FUNCTION_BLOCK "Sequence"   // FB18, GRAPH_PLUS
{ S7_Optimized_Access := 'TRUE' }
VERSION : 0.1
   VAR_INPUT
      OFF_SQ : Bool := false;   // Turn sequence off
      INIT_SQ : Bool := false;   // Set sequence to initial state
      ACK_EF : Bool := false;   // Acknowledge all errors and faults
      S_PREV : Bool := false;   // Output previous step in parameter S_NO
      S_NEXT : Bool := false;   // Indicate next step in parameter S_NO
      SW_AUTO : Bool := false;   // Automatic mode
      SW_TAP : Bool := false;   // Semiautomatic/switch with transition
      SW_TOP : Bool := false;   // Semiautomatic/ignore transition
      SW_MAN : Bool := false;   // Manual mode
      S_SEL : Int := 0;   // Select step to be output to S_NO
      S_ON : Bool := false;   // Activate step indicated in S_NO
      S_OFF : Bool := false;   // Deactivate step indicated S_NO
      T_PUSH : Bool := false;   // Enable transition to switch in semi automatic mode
   END_VAR
   VAR_OUTPUT
      S_NO : Int := 0;   // Step number
      S_MORE : Bool := false;   // More steps are available and can be shown in S_NO
      S_ACTIVE : Bool := false;   // Step indicated in S_NO is active
      ERR_FLT : Bool := false;   // Interlock or supervision group error
      AUTO_ON : Bool := false;   // Automatic mode is active
      TAP_ON : Bool := false;   // Semiautomatic mode/step with transition enabled
      TOP_ON : Bool := false;   // Semiautomatic mode/ignore transition enabled
      MAN_ON : Bool := false;   // Manual mode is active
   END_VAR
   VAR
      HMI_INFO : Array[0..8] of UInt;
      IF_PAR : G7_IfParPlus_V2;
      RT_DATA : G7_RTDataPlus_V2;   // Internal data area
      Trans1 : G7_TransitionPlus_V2;   // Transition structure
      Trans2 : G7_TransitionPlus_V2;   // Transition structure
      Trans3 : G7_TransitionPlus_V2;   // Transition structure
      Trans4 : G7_TransitionPlus_V2;   // Transition structure
      Trans5 : G7_TransitionPlus_V2;   // Transition structure
      idle : G7_StepPlus_V2;   // Step structure
      warmup : G7_StepPlus_V2;   // Step structure
      stabilize : G7_StepPlus_V2;   // Step structure
      Generation : G7_StepPlus_V2;   // Step structure
      cooldown : G7_StepPlus_V2;   // Step structure
      SINI : Array[0..1] of USInt;
      LSTT : Array[0..4] of USInt;
      ATAJ : Array[0..4] of USInt;
      ATAB : Array[0..4] of USInt;
      PSTT : Array[0..4] of USInt;
      NSTT : Array[0..4] of USInt;
      ASSJ : Array[0..4] of USInt;
      ASSB : Array[0..4] of USInt;
      PTTS : Array[0..4] of USInt;
      NTTS : Array[0..4] of USInt;
      SW_SQTS : Array[0..4] of USInt;
      SWITCH : Array[0..0] of USInt;
      TVX : Array[0..1] of USInt;
      TTX : Array[0..1] of USInt;
      TSX : Array[0..1] of USInt;
      S00X : Array[0..1] of USInt;
      SOFFX : Array[0..1] of USInt;
      SONX : Array[0..1] of USInt;
      SAX : Array[0..1] of USInt;
      SERRX : Array[0..5] of USInt;
      SMX : Array[0..5] of USInt;
      S0X : Array[0..5] of USInt;
      S1X : Array[0..5] of USInt;
      IL_ALARM_INST : Program_Alarm;
      SUP_ALARM_INST : Program_Alarm;
      STEP_TIME_ALARM_INST : Program_Alarm;
      IEC_TIMER_INST : IEC_TIMER;
      TRANSACTION_FLAG : Bool := false;
   END_VAR
   // SINI[0] := 2;
   // LSTT[0] := 255;
   // LSTT[1] := 255;
   // LSTT[2] := 255;
   // LSTT[3] := 255;
   // ATAJ[1] := 1;
   // ATAJ[2] := 2;
   // ATAJ[3] := 3;
   // ATAJ[4] := 4;
   // ATAB[1] := 1;
   // ATAB[2] := 2;
   // ATAB[3] := 3;
   // ATAB[4] := 4;
   // PSTT[1] := 1;
   // PSTT[2] := 2;
   // PSTT[3] := 3;
   // PSTT[4] := 4;
   // NSTT[0] := 1;
   // NSTT[1] := 2;
   // NSTT[2] := 3;
   // NSTT[3] := 4;
   // ASSJ[1] := 1;
   // ASSJ[2] := 2;
   // ASSJ[3] := 3;
   // ASSJ[4] := 4;
   // ASSB[1] := 1;
   // ASSB[2] := 2;
   // ASSB[3] := 3;
   // ASSB[4] := 4;
   // PTTS[0] := 255;
   // PTTS[2] := 1;
   // PTTS[3] := 2;
   // PTTS[4] := 3;
   // NTTS[1] := 1;
   // NTTS[2] := 2;
   // NTTS[3] := 3;
   // NTTS[4] := 4;
   // TVX[0] := 16#1;
   // TTX[0] := 16#1;
   // TSX[0] := 16#1;
   // S00X[0] := 16#1;
   // SOFFX[0] := 16#1;
   // SONX[0] := 16#1;
   // SAX[0] := 16#1;
   // SERRX[0] := 16#1;
   // SMX[0] := 16#1;
   // S0X[0] := 16#1;
   // S1X[0] := 16#1;
BEGIN
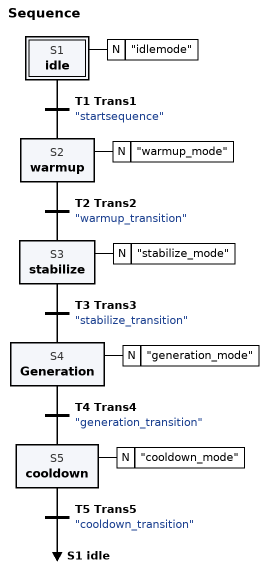
   // sequencer 1
   INITIAL_STEP idle:   // S1, max time T#10S, warning time T#7S
              N    "idlemode"
   END_STEP
   TRANSITION Trans1 FROM idle TO warmup   // T1
      := "startsequence";
   END_TRANSITION
   STEP warmup:   // S2, max time T#10S, warning time T#7S
              N    "warmup_mode"
   END_STEP
   TRANSITION Trans2 FROM warmup TO stabilize   // T2
      := "warmup_transition";
   END_TRANSITION
   STEP stabilize:   // S3, max time T#10S, warning time T#7S
      // stabilize
              N    "stabilize_mode"
   END_STEP
   TRANSITION Trans3 FROM stabilize TO Generation   // T3
      := "stabilize_transition";
   END_TRANSITION
   STEP Generation:   // S4, max time T#10S, warning time T#7S
              N    "generation_mode"
   END_STEP
   TRANSITION Trans4 FROM Generation TO cooldown   // T4
      := "generation_transition";
   END_TRANSITION
   STEP cooldown:   // S5, max time T#10S, warning time T#7S
              N    "cooldown_mode"
   END_STEP
   TRANSITION Trans5 FROM cooldown TO idle   // T5, jump
      := "cooldown_transition";
   END_TRANSITION
END_FUNCTION_BLOCK

FUNCTION_BLOCK "Hourmeter_LAD"   // FB19, LAD
{ S7_Optimized_Access := 'TRUE' }
VERSION : 0.1
   VAR
      onsh1 : Bool;
      onsh2 : Bool;
      onsh3 : Bool;
      onsh4 : Bool;
      onsh5 : Bool;
   END_VAR
   VAR_TEMP   // added for the SCL form of the ladder/FBD networks
      _w1 : Bool;
      _w2 : Bool;
      _w3 : Bool;
   END_VAR
BEGIN

REGION Network 1
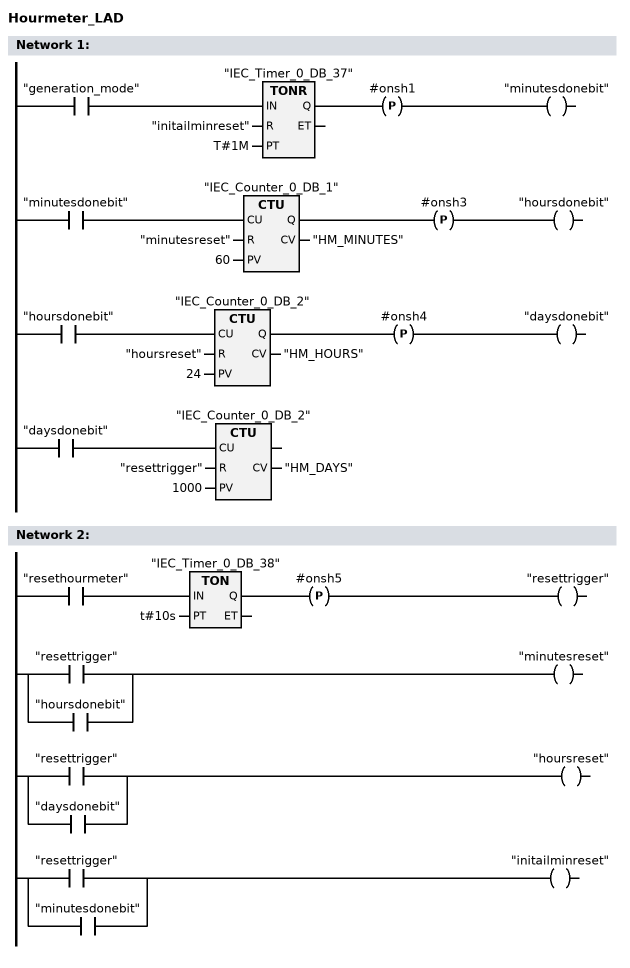
   "IEC_Timer_0_DB_37".TONR(IN := "generation_mode", R := "initailminreset", PT := T#1M);
   #_w1 := "IEC_Timer_0_DB_37".Q AND NOT #onsh1;   // rising edge
   #onsh1 := "IEC_Timer_0_DB_37".Q;
   "minutesdonebit" := #_w1;
   "IEC_Counter_0_DB_1".CTU(CU := "minutesdonebit", R := "minutesreset", PV := 60, CV => "HM_MINUTES");
   #_w2 := "IEC_Counter_0_DB_1".Q AND NOT #onsh3;   // rising edge
   #onsh3 := "IEC_Counter_0_DB_1".Q;
   "hoursdonebit" := #_w2;
   "IEC_Counter_0_DB_2".CTU(CU := "hoursdonebit", R := "hoursreset", PV := 24, CV => "HM_HOURS");
   #_w3 := "IEC_Counter_0_DB_2".Q AND NOT #onsh4;   // rising edge
   #onsh4 := "IEC_Counter_0_DB_2".Q;
   "daysdonebit" := #_w3;
   "IEC_Counter_0_DB_2".CTU(CU := "daysdonebit", R := "resettrigger", PV := 1000, CV => "HM_DAYS");
END_REGION

REGION Network 2
   "IEC_Timer_0_DB_38".TON(IN := "resethourmeter", PT := t#10s);
   #_w1 := "IEC_Timer_0_DB_38".Q AND NOT #onsh5;   // rising edge
   #onsh5 := "IEC_Timer_0_DB_38".Q;
   "resettrigger" := #_w1;
   "minutesreset" := "resettrigger" OR "hoursdonebit";
   "hoursreset" := "resettrigger" OR "daysdonebit";
   "initailminreset" := "resettrigger" OR "minutesdonebit";
END_REGION
END_FUNCTION_BLOCK

FUNCTION_BLOCK "HOURMETER_FBD"   // FB20, FBD
{ S7_Optimized_Access := 'TRUE' }
VERSION : 0.1
   VAR
      onsh1 : Bool;
      onsh2 : Bool;
      onsh3 : Bool;
      onsh4 : Bool;
   END_VAR
   VAR_TEMP   // added for the SCL form of the ladder/FBD networks
      _w1 : Bool;
      _w2 : Bool;
      _w3 : Bool;
   END_VAR
BEGIN

REGION Network 1
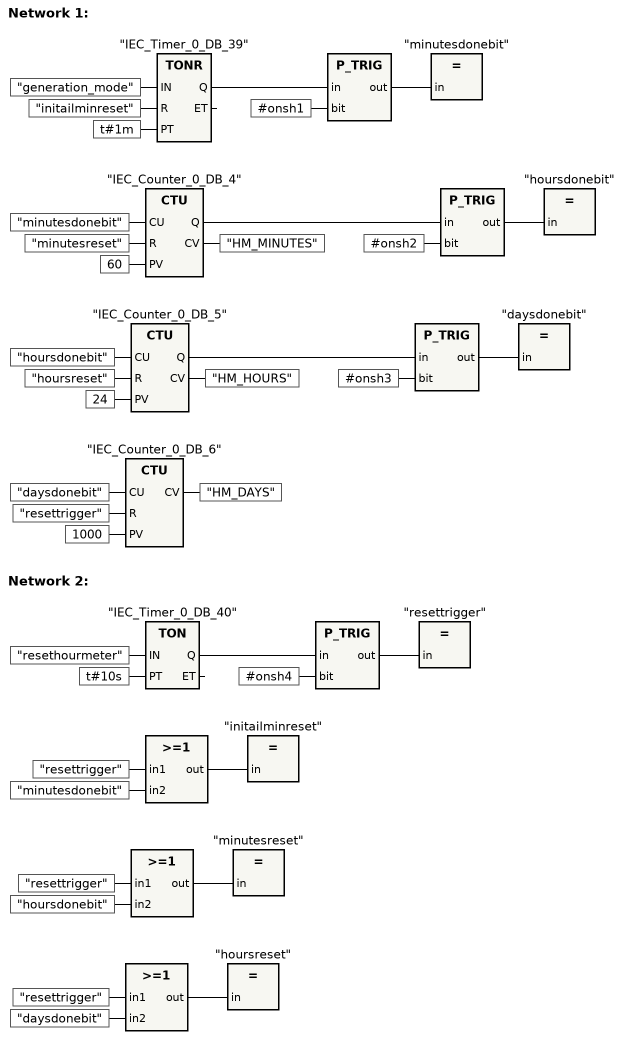
   "IEC_Timer_0_DB_39".TONR(IN := "generation_mode", R := "initailminreset", PT := t#1m);
   #_w1 := "IEC_Timer_0_DB_39".Q AND NOT #onsh1;   // rising edge
   #onsh1 := "IEC_Timer_0_DB_39".Q;
   "minutesdonebit" := #_w1;
   "IEC_Counter_0_DB_4".CTU(CU := "minutesdonebit", R := "minutesreset", PV := 60, CV => "HM_MINUTES");
   #_w2 := "IEC_Counter_0_DB_4".Q AND NOT #onsh2;   // rising edge
   #onsh2 := "IEC_Counter_0_DB_4".Q;
   "hoursdonebit" := #_w2;
   "IEC_Counter_0_DB_5".CTU(CU := "hoursdonebit", R := "hoursreset", PV := 24, CV => "HM_HOURS");
   #_w3 := "IEC_Counter_0_DB_5".Q AND NOT #onsh3;   // rising edge
   #onsh3 := "IEC_Counter_0_DB_5".Q;
   "daysdonebit" := #_w3;
   "IEC_Counter_0_DB_6".CTU(CU := "daysdonebit", R := "resettrigger", PV := 1000, CV => "HM_DAYS");
END_REGION

REGION Network 2
   "IEC_Timer_0_DB_40".TON(IN := "resethourmeter", PT := t#10s);
   #_w1 := "IEC_Timer_0_DB_40".Q AND NOT #onsh4;   // rising edge
   #onsh4 := "IEC_Timer_0_DB_40".Q;
   "resettrigger" := #_w1;
   "initailminreset" := "resettrigger" OR "minutesdonebit";
   "minutesreset" := "resettrigger" OR "hoursdonebit";
   "hoursreset" := "resettrigger" OR "daysdonebit";
END_REGION
END_FUNCTION_BLOCK

FUNCTION_BLOCK "HOURMETER_SCL"   // FB21, SCL
{ S7_Optimized_Access := 'TRUE' }
VERSION : 0.1
   VAR
      trigger1 : Bool;
      onsh1 : Bool;
      onsh1trigger : Bool;
   END_VAR
   VAR_TEMP
      t11 : Time;
      daysss : Bool;
      TT2 : Time;
   END_VAR
BEGIN
   IF "generation_mode" THEN
       "IEC_Timer_0_DB_42".TONR(IN := TRUE,
                                R := "initailminreset",
                                PT := T#1M,
                                Q => "minutesdonebit",
                                ET => #t11);
   END_IF;

   IF "minutesdonebit" THEN
       RESET_TIMER("IEC_Timer_0_DB_42");
   END_IF;

   "IEC_Counter_0_DB_7".CTU(CU := "minutesdonebit",
                                R := "minutesreset",
                                PV := 60,
                                Q => "hoursdonebit",
                                CV => "HM_MINUTES");



       "IEC_Counter_0_DB_8".CTU(CU := "hoursdonebit",
                                R := "hoursreset",
                                PV := 24,
                                Q => "daysdonebit",
                                CV => "HM_HOURS");



       "IEC_Counter_0_DB_9".CTU(CU := "daysdonebit",
                                R := "resettrigger",
                                PV := 10000,
                                Q => #daysss,
                                CV => "HM_DAYS");



   IF "resethourmeter"  THEN
       "IEC_Timer_0_DB_44".TON(IN:=TRUE,
                               PT:=T#10S,
                               Q=>"resettrigger",
                               ET=>#TT2);
   ELSE
      RESET_TIMER("IEC_Timer_0_DB_44");
      "resettrigger" := 0;
   END_IF;

   IF "resettrigger" OR "minutesdonebit" THEN
       "initailminreset" := 1;
   ELSE
       "initailminreset" := 0;

   END_IF;

   IF "resettrigger" OR "hoursdonebit" THEN
       "minutesreset" := 1;
   ELSE
        "minutesreset" := 0;

   END_IF;


   IF "resettrigger" OR "daysdonebit" THEN
       "hoursreset" := 1;
   ELSE
       "hoursreset" := 0;

   END_IF;
END_FUNCTION_BLOCK

FUNCTION_BLOCK "HOURMETER_STL"   // FB22, STL
{ S7_Optimized_Access := 'TRUE' }
VERSION : 0.1
   VAR_TEMP
      TT1 : Time;
      TT2 : Time;
      DAYSSS : Bool;
   END_VAR
BEGIN

REGION Network 1
         A     "generation_mode";
         JC    timerRTO;
         CLR;

         JU    endofline;

   timerRTO:CALL  TONR , "IEC_Timer_0_DB_43"
         ( IN := TRUE,
           R  := "initailminreset",
           PT := T#60S,
           Q  := "minutesdonebit",
           ET := #TT1
         );

         CALL  CTU, "IEC_Counter_0_DB_10"
         ( CU := "minutesdonebit",
           R  := "minutesreset",
           PV := 60,
           Q  := "hoursdonebit",
           CV := "HM_MINUTES"
         );


         CALL  CTU, "IEC_Counter_0_DB_11"
         ( CU := "hoursdonebit",
           R  := "hoursreset",
           PV := 24,
           Q  := "daysdonebit",
           CV := "HM_HOURS"
         );

         CALL  CTU, "IEC_Counter_0_DB_12"
         ( CU := "daysdonebit",
           R  := "resettrigger",
           PV := 1000,
           Q  := #DAYSSS,
           CV := "HM_DAYS"
         );

         JU    reset;

   reset:CLR;
         A     "resethourmeter";
         JC    resethourmeter;
         CALL  RESET_TIMER
         ( "TIMER" := "IEC_Timer_0_DB_45"
         );
         JU    endofline;

   resethourmeter:CALL  TON, "IEC_Timer_0_DB_45"
         ( IN := TRUE,
           PT := T#10S,
           Q  := "resettrigger",
           ET := #TT2
         );
         A     "resettrigger";
         JU    endofline;


   endofline:CLR;



         A     "resettrigger";
         O     "minutesdonebit";
         =     "initailminreset";
         CLR;
         A     "resettrigger";
         O     "hoursdonebit";
         =     "minutesreset";
         CLR;
         A     "resettrigger";
         O     "daysdonebit";
         =     "hoursreset";
END_REGION
END_FUNCTION_BLOCK

FUNCTION "Scalingblock" : Void   // FC1, FBD
{ S7_Optimized_Access := 'TRUE' }
VERSION : 0.1
   VAR_INPUT
      intput_min : DInt;
      input_max : Int;
      output_min : Int;
      output_max : Int;
      input_value : Int;
   END_VAR
   VAR_OUTPUT
      sv : Int;
   END_VAR
   VAR_TEMP
      input_min : Int;
      tv : Real;
   END_VAR
BEGIN

REGION Network 1
   // scaling
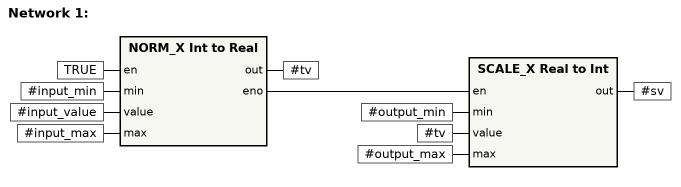
   IF TRUE THEN
       #tv := NORM_X(MIN := #input_min, VALUE := #input_value, MAX := #input_max);
       #sv := SCALE_X(MIN := #output_min, VALUE := #tv, MAX := #output_max);
   END_IF;
END_REGION
END_FUNCTION

FUNCTION "CONVERTTIME" : Void   // FC2, FBD
{ S7_Optimized_Access := 'TRUE' }
VERSION : 0.1
   VAR_INPUT
      VALUEIN : Int;
   END_VAR
   VAR_OUTPUT
      Time1 : Time;
   END_VAR
   VAR_TEMP
      TTV1 : Int;
   END_VAR
BEGIN

REGION Network 1
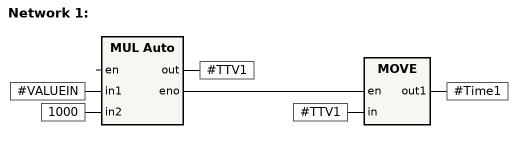
   #TTV1 := #VALUEIN * 1000;
   #Time1 := #TTV1;
END_REGION
END_FUNCTION

ORGANIZATION_BLOCK "Main"   // OB1, LAD, ProgramCycle
TITLE = "Main Program Sweep (Cycle)"
{ S7_Optimized_Access := 'TRUE' }
VERSION : 0.1
   VAR_INPUT
      Initial_Call : Bool;   // Initial call of this OB
      Remanence : Bool;   // =True, if remanent data are available
   END_VAR
   VAR_TEMP
      SequenceInit : Bool;
      InitSequence : Bool;
   END_VAR
   VAR_TEMP   // added for the SCL form of the ladder/FBD networks
      _w1 : Bool;
      _w2 : Bool;
      _w3 : Bool;
      _w4 : Bool;
   END_VAR
BEGIN

REGION Network 1
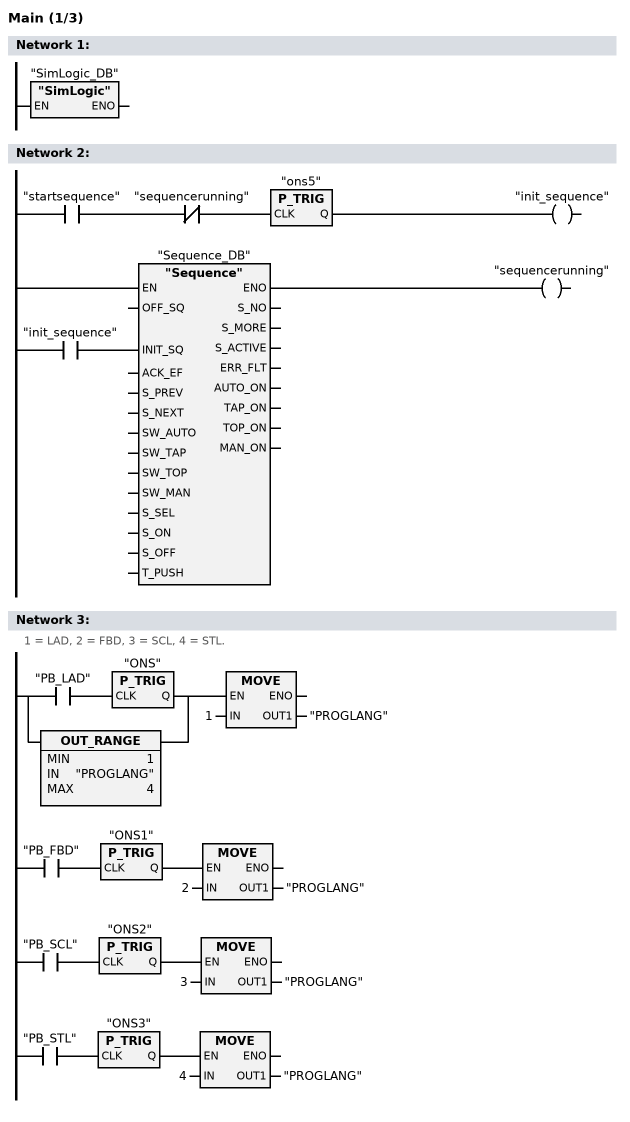
   RUNG wire#powerrail
      "SimLogic_DB"()
   END_RUNG
   // the same network as SCL:
   "SimLogic_DB"();   // "SimLogic"
END_REGION

REGION Network 2
   RUNG wire#powerrail
      Contact( "startsequence" )
      I_Contact( "sequencerunning" )
      P_Trig( "ons5" )
      Coil( "init_sequence" )
   END_RUNG
   RUNG wire#powerrail
      "Sequence_DB"(INIT_SQ := wire#w1, OFF_SQ :=, ACK_EF :=, S_PREV :=, S_NEXT :=, SW_AUTO :=, SW_TAP :=, SW_TOP :=, SW_MAN :=, S_SEL :=, S_ON :=, S_OFF :=, T_PUSH :=, S_NO =>, S_MORE =>, S_ACTIVE =>, ERR_FLT =>, AUTO_ON =>, TAP_ON =>, TOP_ON =>, MAN_ON =>)
      Coil( "sequencerunning" )
   END_RUNG
   RUNG wire#powerrail
      Contact( "init_sequence" )
   END_RUNG wire#w1
   // the same network as SCL:
   #_w1 := "startsequence" AND NOT "sequencerunning";
   #_w2 := #_w1 AND NOT "ons5";   // rising edge
   "ons5" := #_w1;
   "init_sequence" := #_w2;
   "Sequence_DB"(INIT_SQ := "init_sequence", ENO => #_w3);   // "Sequence"
   "sequencerunning" := #_w3;
END_REGION

REGION Network 3
   // 1 = LAD, 2 = FBD, 3 = SCL, 4 = STL.
   #_w1 := "PB_LAD" AND NOT "ONS";   // rising edge
   "ONS" := "PB_LAD";
   IF #_w1 OR ("PROGLANG" < 1) OR ("PROGLANG" > 4) THEN "PROGLANG" := 1; END_IF;
   #_w2 := "PB_FBD" AND NOT "ONS1";   // rising edge
   "ONS1" := "PB_FBD";
   IF #_w2 THEN "PROGLANG" := 2; END_IF;
   #_w3 := "PB_SCL" AND NOT "ONS2";   // rising edge
   "ONS2" := "PB_SCL";
   IF #_w3 THEN "PROGLANG" := 3; END_IF;
   #_w4 := "PB_STL" AND NOT "ONS3";   // rising edge
   "ONS3" := "PB_STL";
   IF #_w4 THEN "PROGLANG" := 4; END_IF;
END_REGION

REGION Network 4
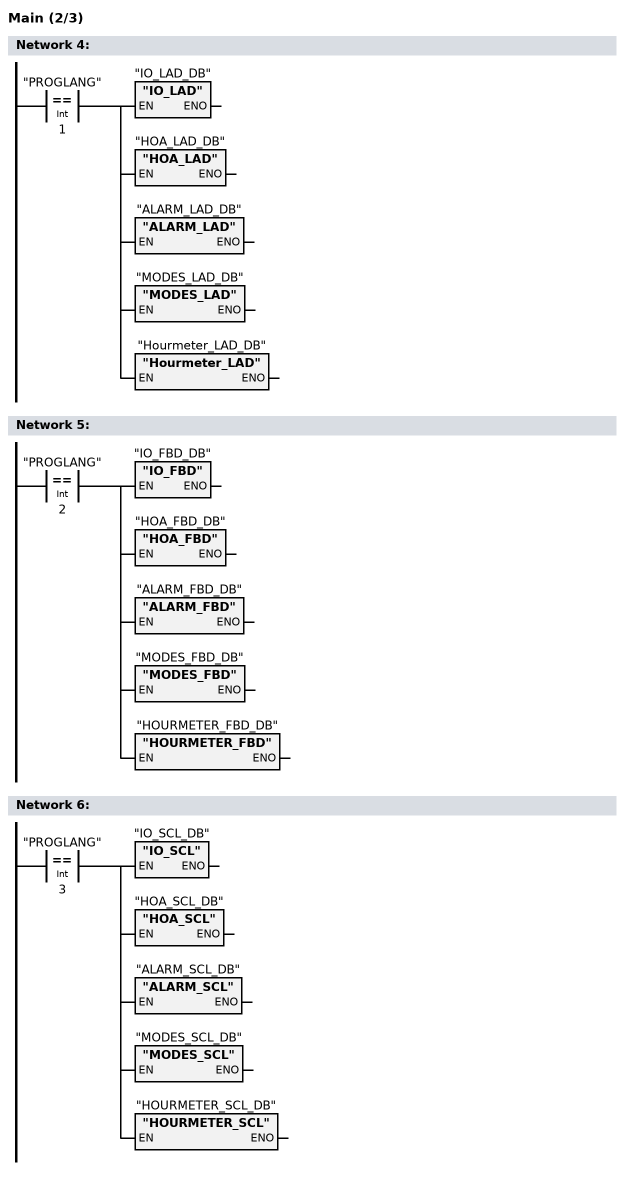
   RUNG wire#powerrail
      { S7_Templates := "SrcType := Int" } EQ_Contact(in1 := "PROGLANG", in2 := 1)
      wire#w1
      "IO_LAD_DB"()
   END_RUNG
   RUNG wire#w1
      "HOA_LAD_DB"()
   END_RUNG
   RUNG wire#w1
      "ALARM_LAD_DB"()
   END_RUNG
   RUNG wire#w1
      "MODES_LAD_DB"()
   END_RUNG
   RUNG wire#w1
      "Hourmeter_LAD_DB"()
   END_RUNG
   // the same network as SCL:
   #_w1 := "PROGLANG" = 1;
   IF #_w1 THEN
       "IO_LAD_DB"();   // "IO_LAD"
       "HOA_LAD_DB"();   // "HOA_LAD"
       "ALARM_LAD_DB"();   // "ALARM_LAD"
       "MODES_LAD_DB"();   // "MODES_LAD"
       "Hourmeter_LAD_DB"();   // "Hourmeter_LAD"
   END_IF;
END_REGION

REGION Network 5
   RUNG wire#powerrail
      { S7_Templates := "SrcType := Int" } EQ_Contact(in1 := "PROGLANG", in2 := 2)
      wire#w1
      "IO_FBD_DB"()
   END_RUNG
   RUNG wire#w1
      "HOA_FBD_DB"()
   END_RUNG
   RUNG wire#w1
      "ALARM_FBD_DB"()
   END_RUNG
   RUNG wire#w1
      "MODES_FBD_DB"()
   END_RUNG
   RUNG wire#w1
      "HOURMETER_FBD_DB"()
   END_RUNG
   // the same network as SCL:
   #_w1 := "PROGLANG" = 2;
   IF #_w1 THEN
       "IO_FBD_DB"();   // "IO_FBD"
       "HOA_FBD_DB"();   // "HOA_FBD"
       "ALARM_FBD_DB"();   // "ALARM_FBD"
       "MODES_FBD_DB"();   // "MODES_FBD"
       "HOURMETER_FBD_DB"();   // "HOURMETER_FBD"
   END_IF;
END_REGION

REGION Network 6
   RUNG wire#powerrail
      { S7_Templates := "SrcType := Int" } EQ_Contact(in1 := "PROGLANG", in2 := 3)
      wire#w1
      "IO_SCL_DB"()
   END_RUNG
   RUNG wire#w1
      "HOA_SCL_DB"()
   END_RUNG
   RUNG wire#w1
      "ALARM_SCL_DB"()
   END_RUNG
   RUNG wire#w1
      "MODES_SCL_DB"()
   END_RUNG
   RUNG wire#w1
      "HOURMETER_SCL_DB"()
   END_RUNG
   // the same network as SCL:
   #_w1 := "PROGLANG" = 3;
   IF #_w1 THEN
       "IO_SCL_DB"();   // "IO_SCL"
       "HOA_SCL_DB"();   // "HOA_SCL"
       "ALARM_SCL_DB"();   // "ALARM_SCL"
       "MODES_SCL_DB"();   // "MODES_SCL"
       "HOURMETER_SCL_DB"();   // "HOURMETER_SCL"
   END_IF;
END_REGION

REGION Network 7
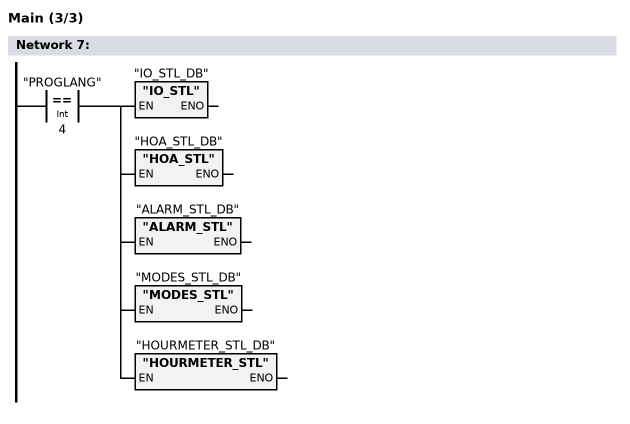
   RUNG wire#powerrail
      { S7_Templates := "SrcType := Int" } EQ_Contact(in1 := "PROGLANG", in2 := 4)
      wire#w1
      "IO_STL_DB"()
   END_RUNG
   RUNG wire#w1
      "HOA_STL_DB"()
   END_RUNG
   RUNG wire#w1
      "ALARM_STL_DB"()
   END_RUNG
   RUNG wire#w1
      "MODES_STL_DB"()
   END_RUNG
   RUNG wire#w1
      "HOURMETER_STL_DB"()
   END_RUNG
   // the same network as SCL:
   #_w1 := "PROGLANG" = 4;
   IF #_w1 THEN
       "IO_STL_DB"();   // "IO_STL"
       "HOA_STL_DB"();   // "HOA_STL"
       "ALARM_STL_DB"();   // "ALARM_STL"
       "MODES_STL_DB"();   // "MODES_STL"
       "HOURMETER_STL_DB"();   // "HOURMETER_STL"
   END_IF;
END_REGION
END_ORGANIZATION_BLOCK

ORGANIZATION_BLOCK "PID"   // OB30, LAD, CyclicInterrupt
{ S7_Optimized_Access := 'TRUE' }
VERSION : 0.1
   VAR_INPUT
      Initial_Call : Bool;   // Initial call of this OB
      Event_Count : Int;   // Events discarded
   END_VAR
   VAR_TEMP
      BSP : Real;
      VSP : Real;
      bafflehandtrigger : Bool;
      baffleofftrigger : Bool;
      baffleautotrigger : Bool;
      vfdhandtrigger : Bool;
      vfdofftrigger : Bool;
      vfdautotrigger : Bool;
   END_VAR
   VAR_TEMP   // added for the SCL form of the ladder/FBD networks
      _w1 : Bool;
      _w2 : Bool;
      _w3 : Bool;
      _w4 : Bool;
      _w5 : Bool;
      _w6 : Bool;
      _w7 : Bool;
   END_VAR
BEGIN

REGION Network 1
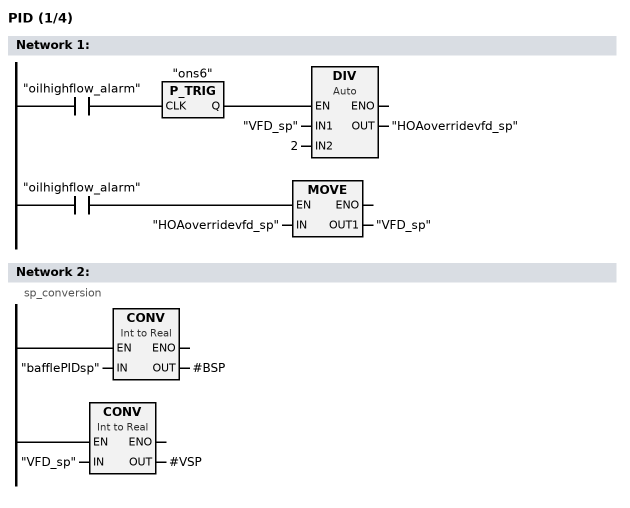
   RUNG wire#powerrail
      Contact( "oilhighflow_alarm" )
      P_Trig( "ons6" )
      Div(in1 := "VFD_sp", in2 := 2, out => "HOAoverridevfd_sp")
   END_RUNG
   RUNG wire#powerrail
      Contact( "oilhighflow_alarm" )
      Move(in := "HOAoverridevfd_sp", out1 => "VFD_sp")
   END_RUNG
   // the same network as SCL:
   #_w1 := "oilhighflow_alarm" AND NOT "ons6";   // rising edge
   "ons6" := "oilhighflow_alarm";
   IF #_w1 THEN "HOAoverridevfd_sp" := "VFD_sp" / 2; END_IF;
   IF "oilhighflow_alarm" THEN "VFD_sp" := "HOAoverridevfd_sp"; END_IF;
END_REGION

REGION Network 2
   // sp_conversion
   RUNG wire#powerrail
      { S7_Templates := "[SrcType := Int, DestType := Real]" } Convert(in := "bafflePIDsp", out => #BSP)
   END_RUNG
   RUNG wire#powerrail
      { S7_Templates := "[SrcType := Int, DestType := Real]" } Convert(in := "VFD_sp", out => #VSP)
   END_RUNG
   // the same network as SCL:
   #BSP := INT_TO_REAL("bafflePIDsp");
   #VSP := INT_TO_REAL("VFD_sp");
END_REGION

REGION Network 3
   // baffle hoa and I/0
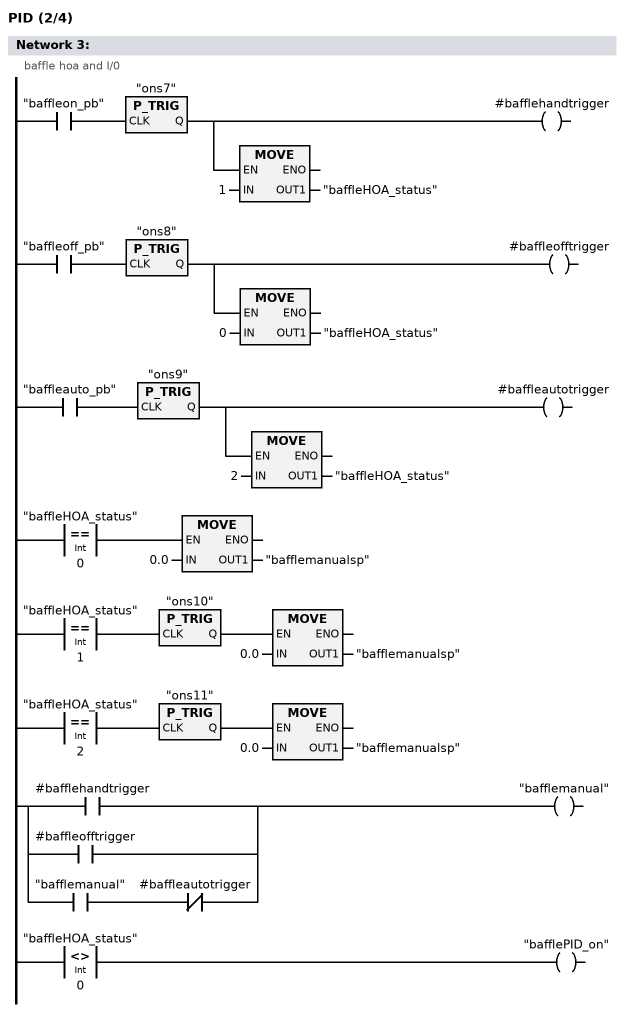
   RUNG wire#powerrail
      Contact( "baffleon_pb" )
      P_Trig( "ons7" )
      wire#w1
      Coil( #bafflehandtrigger )
   END_RUNG
   RUNG wire#w1
      Move(in := 1, out1 => "baffleHOA_status")
   END_RUNG
   RUNG wire#powerrail
      Contact( "baffleoff_pb" )
      P_Trig( "ons8" )
      wire#w2
      Coil( #baffleofftrigger )
   END_RUNG
   RUNG wire#w2
      Move(in := 0, out1 => "baffleHOA_status")
   END_RUNG
   RUNG wire#powerrail
      Contact( "baffleauto_pb" )
      P_Trig( "ons9" )
      wire#w3
      Coil( #baffleautotrigger )
   END_RUNG
   RUNG wire#w3
      Move(in := 2, out1 => "baffleHOA_status")
   END_RUNG
   RUNG wire#powerrail
      { S7_Templates := "SrcType := Int" } EQ_Contact(in1 := "baffleHOA_status", in2 := 0)
      Move(in := 0.0, out1 => "bafflemanualsp")
   END_RUNG
   RUNG wire#powerrail
      { S7_Templates := "SrcType := Int" } EQ_Contact(in1 := "baffleHOA_status", in2 := 1)
      P_Trig( "ons10" )
      Move(in := 0.0, out1 => "bafflemanualsp")
   END_RUNG
   RUNG wire#powerrail
      { S7_Templates := "SrcType := Int" } EQ_Contact(in1 := "baffleHOA_status", in2 := 2)
      P_Trig( "ons11" )
      Move(in := 0.0, out1 => "bafflemanualsp")
   END_RUNG
   RUNG wire#powerrail
      Contact( #bafflehandtrigger )
      wire#w4
      Coil( "bafflemanual" )
   END_RUNG
   RUNG wire#powerrail
      Contact( #baffleofftrigger )
   END_RUNG wire#w4
   RUNG wire#powerrail
      Contact( "bafflemanual" )
      I_Contact( #baffleautotrigger )
   END_RUNG wire#w4
   RUNG wire#powerrail
      { S7_Templates := "SrcType := Int" } NE_Contact(in1 := "baffleHOA_status", in2 := 0)
      Coil( "bafflePID_on" )
   END_RUNG
   // the same network as SCL:
   #_w1 := "baffleon_pb" AND NOT "ons7";   // rising edge
   "ons7" := "baffleon_pb";
   #bafflehandtrigger := #_w1;
   IF #_w1 THEN "baffleHOA_status" := 1; END_IF;
   #_w2 := "baffleoff_pb" AND NOT "ons8";   // rising edge
   "ons8" := "baffleoff_pb";
   #baffleofftrigger := #_w2;
   IF #_w2 THEN "baffleHOA_status" := 0; END_IF;
   #_w3 := "baffleauto_pb" AND NOT "ons9";   // rising edge
   "ons9" := "baffleauto_pb";
   #baffleautotrigger := #_w3;
   IF #_w3 THEN "baffleHOA_status" := 2; END_IF;
   IF "baffleHOA_status" = 0 THEN "bafflemanualsp" := 0.0; END_IF;
   #_w4 := "baffleHOA_status" = 1;
   #_w5 := #_w4 AND NOT "ons10";   // rising edge
   "ons10" := #_w4;
   IF #_w5 THEN "bafflemanualsp" := 0.0; END_IF;
   #_w6 := "baffleHOA_status" = 2;
   #_w7 := #_w6 AND NOT "ons11";   // rising edge
   "ons11" := #_w6;
   IF #_w7 THEN "bafflemanualsp" := 0.0; END_IF;
   "bafflemanual" := #bafflehandtrigger OR #baffleofftrigger OR ("bafflemanual" AND NOT #baffleautotrigger);
   "bafflePID_on" := "baffleHOA_status" <> 0;
END_REGION

REGION Network 4
   // vfd hoa and I/0
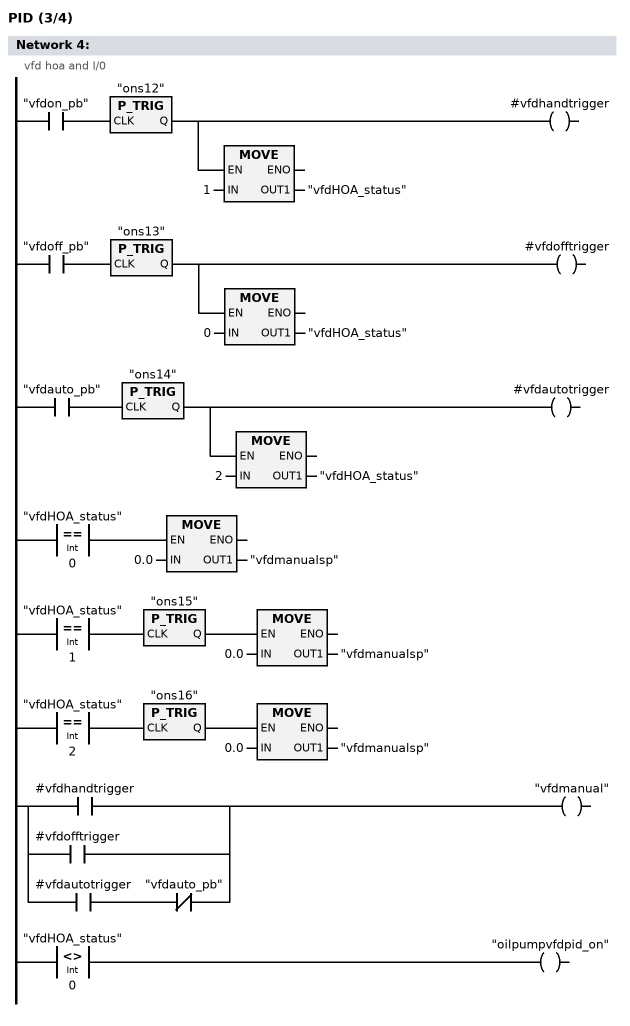
   RUNG wire#powerrail
      Contact( "vfdon_pb" )
      P_Trig( "ons12" )
      wire#w1
      Coil( #vfdhandtrigger )
   END_RUNG
   RUNG wire#w1
      Move(in := 1, out1 => "vfdHOA_status")
   END_RUNG
   RUNG wire#powerrail
      Contact( "vfdoff_pb" )
      P_Trig( "ons13" )
      wire#w2
      Coil( #vfdofftrigger )
   END_RUNG
   RUNG wire#w2
      Move(in := 0, out1 => "vfdHOA_status")
   END_RUNG
   RUNG wire#powerrail
      Contact( "vfdauto_pb" )
      P_Trig( "ons14" )
      wire#w3
      Coil( #vfdautotrigger )
   END_RUNG
   RUNG wire#w3
      Move(in := 2, out1 => "vfdHOA_status")
   END_RUNG
   RUNG wire#powerrail
      { S7_Templates := "SrcType := Int" } EQ_Contact(in1 := "vfdHOA_status", in2 := 0)
      Move(in := 0.0, out1 => "vfdmanualsp")
   END_RUNG
   RUNG wire#powerrail
      { S7_Templates := "SrcType := Int" } EQ_Contact(in1 := "vfdHOA_status", in2 := 1)
      P_Trig( "ons15" )
      Move(in := 0.0, out1 => "vfdmanualsp")
   END_RUNG
   RUNG wire#powerrail
      { S7_Templates := "SrcType := Int" } EQ_Contact(in1 := "vfdHOA_status", in2 := 2)
      P_Trig( "ons16" )
      Move(in := 0.0, out1 => "vfdmanualsp")
   END_RUNG
   RUNG wire#powerrail
      Contact( #vfdhandtrigger )
      wire#w4
      Coil( "vfdmanual" )
   END_RUNG
   RUNG wire#powerrail
      Contact( #vfdofftrigger )
   END_RUNG wire#w4
   RUNG wire#powerrail
      Contact( #vfdautotrigger )
      I_Contact( "vfdauto_pb" )
   END_RUNG wire#w4
   RUNG wire#powerrail
      { S7_Templates := "SrcType := Int" } NE_Contact(in1 := "vfdHOA_status", in2 := 0)
      Coil( "oilpumpvfdpid_on" )
   END_RUNG
   // the same network as SCL:
   #_w1 := "vfdon_pb" AND NOT "ons12";   // rising edge
   "ons12" := "vfdon_pb";
   #vfdhandtrigger := #_w1;
   IF #_w1 THEN "vfdHOA_status" := 1; END_IF;
   #_w2 := "vfdoff_pb" AND NOT "ons13";   // rising edge
   "ons13" := "vfdoff_pb";
   #vfdofftrigger := #_w2;
   IF #_w2 THEN "vfdHOA_status" := 0; END_IF;
   #_w3 := "vfdauto_pb" AND NOT "ons14";   // rising edge
   "ons14" := "vfdauto_pb";
   #vfdautotrigger := #_w3;
   IF #_w3 THEN "vfdHOA_status" := 2; END_IF;
   IF "vfdHOA_status" = 0 THEN "vfdmanualsp" := 0.0; END_IF;
   #_w4 := "vfdHOA_status" = 1;
   #_w5 := #_w4 AND NOT "ons15";   // rising edge
   "ons15" := #_w4;
   IF #_w5 THEN "vfdmanualsp" := 0.0; END_IF;
   #_w6 := "vfdHOA_status" = 2;
   #_w7 := #_w6 AND NOT "ons16";   // rising edge
   "ons16" := #_w6;
   IF #_w7 THEN "vfdmanualsp" := 0.0; END_IF;
   "vfdmanual" := #vfdhandtrigger OR #vfdofftrigger OR (#vfdautotrigger AND NOT "vfdauto_pb");
   "oilpumpvfdpid_on" := "vfdHOA_status" <> 0;
END_REGION

REGION Network 5
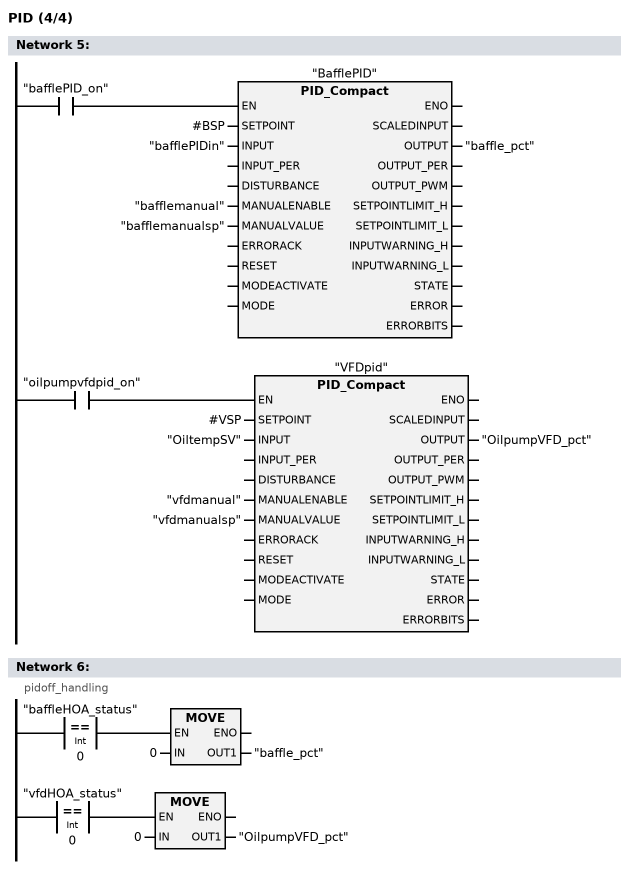
   IF "bafflePID_on" THEN
       "BafflePID"(Setpoint := #BSP,   // PID_Compact
                   Input := "bafflePIDin",
                   ManualEnable := "bafflemanual",
                   ManualValue := "bafflemanualsp",
                   Output => "baffle_pct");
   END_IF;
   IF "oilpumpvfdpid_on" THEN
       "VFDpid"(Setpoint := #VSP,   // PID_Compact
                Input := "OiltempSV",
                ManualEnable := "vfdmanual",
                ManualValue := "vfdmanualsp",
                Output => "OilpumpVFD_pct");
   END_IF;
END_REGION

REGION Network 6
   // pidoff_handling
   RUNG wire#powerrail
      { S7_Templates := "SrcType := Int" } EQ_Contact(in1 := "baffleHOA_status", in2 := 0)
      Move(in := 0, out1 => "baffle_pct")
   END_RUNG
   RUNG wire#powerrail
      { S7_Templates := "SrcType := Int" } EQ_Contact(in1 := "vfdHOA_status", in2 := 0)
      Move(in := 0, out1 => "OilpumpVFD_pct")
   END_RUNG
   // the same network as SCL:
   IF "baffleHOA_status" = 0 THEN "baffle_pct" := 0; END_IF;
   IF "vfdHOA_status" = 0 THEN "OilpumpVFD_pct" := 0; END_IF;
END_REGION
END_ORGANIZATION_BLOCK

(* ===== HMI "HMI_RT_1" =====
system functions are stored by id; their names below are inferred from use
connection "HMI_Connection_1": ETHERNET, S7_1500_OMS

HMI tags "Default tag table"
   "systemstart_pb" : Bool = PLC systemstart_pb AT %M53.0, 1 s
   "systemstop_pb" : Bool = PLC systemstop_pb AT %M53.3, 1 s
   "E-stop_alarm" : Bool = PLC "E-STOP_ALARM" AT %M74.3, 1 s
   "brakefailurealarm" : Bool = PLC brakefailure_alarm AT %M33.5, 1 s
   "highoilflow_alarm" : Bool = PLC oilhighflow_alarm AT %M33.4, 1 s
   "lowoilflow_alarm" : Bool = PLC oillowflow_alarm AT %M33.1, 1 s
   "highoiltemp_alarm" : Bool = PLC oilhightemp_alarm AT %M48.6, 1 s
   "overspeedalarm" : Bool = PLC RPM_ALM AT %M33.3, 1 s
   "overcurrentalarm" : Bool = PLC overcurrent_alarm AT %M33.2, 1 s
   "alarmsilence" : Bool = PLC alarm_rst_notify AT %M48.1, 1 s
   "alarmreset" : Bool = PLC Alarm_reset AT %M35.5, 1 s
   "brakeEn" : Bool = PLC Brake_Out AT %M0.0, 1 s
   "stationinterlockEn" : Bool = PLC stationInterlock_out AT %M1.4, 1 s
   "vfdEn" : Bool = PLC OilPumpVFDen_Out AT %M0.2, 1 s
   "baffleEn" : Bool = PLC Baffle_En AT %M0.1, 1 s
   "alarmhornEn" : Bool = PLC AlarmHorn_out AT %M1.3, 1 s
   "brakehandpb" : Bool = PLC brakeon_pb AT %M34.1, 1 s
   "brakeoffpb" : Bool = PLC brakeoff_pb AT %M34.0, 1 s
   "brakeautopb" : Bool = PLC brakeauto_pb AT %M34.2, 1 s
   "stationinterlockhandpb" : Bool = PLC stationinterlockon_pb AT %M34.7, 1 s
   "stationinterlockoffpb" : Bool = PLC stationinterlockoff_pb AT %M34.6, 1 s
   "stationinterlockautopb" : Bool = PLC stationinterlockauto_pb AT %M35.0, 1 s
   "vfdhandpb" : Bool = PLC vfdon_pb AT %M110.1, 1 s
   "vfdoffpb" : Bool = PLC vfdoff_pb AT %M110.7, 1 s
   "vfdautopb" : Bool = PLC vfdauto_pb AT %M111.0, 1 s
   "bafflehandpb" : Bool = PLC baffleon_pb AT %M52.2, 1 s
   "baffleoffpb" : Bool = PLC baffleoff_pb AT %M75.2, 1 s
   "baffleautopb" : Bool = PLC baffleauto_pb AT %M52.1, 1 s
   "alarmhornhandpb" : Bool = PLC alarmhornon_pb AT %M34.4, 1 s
   "alarmhornoffpb" : Bool = PLC alarmhornoff_pb AT %M34.3, 1 s
   "alarmhornautopb" : Bool = PLC alarmhornauto_pb AT %M34.5, 1 s
   "brakehoa" : Int = PLC brakeHOA_status AT %MW36, 1 s
   "stationinterlockhoa" : Int = PLC stationinterlockHOA_status AT %MW40, 1 s
   "vfdhoa" : Int = PLC vfdHOA_status AT %MW112, 1 s
   "alarmhornhoa" : Int = PLC alarmhornHOA_status AT %MW38, 1 s
   "bafflehoa" : Int = PLC baffleHOA_status AT %MW42, 1 s
   "HM_minutes" : Int = PLC HM_MINUTES AT %MW118, 1 s
   "HM_hours" : Int = PLC HM_HOURS AT %MW120, 1 s
   "HM_days" : Int = PLC HM_DAYS AT %MW122, 1 s
   "hourmetereset_pb" : Bool = PLC resethourmeter AT %M32.5, 1 s
   "faultmode" : Bool = PLC faultmode AT %M53.7, 1 s
   "brakefailuredelay" : Int = PLC brakefailuredelay_SP AT %MW72, 1 s
   "overcurrrentsp" : Int = PLC overcurrent_SP AT %MW50, 1 s
   "overcurrentdelay" : Int = PLC overcurrentdelya_SP AT %MW54, 1 s
   "overspeedsp" : Int = PLC RPM_SP AT %MW66, 1 s
   "overspeeddelay" : Int = PLC rotoroverspeeddelay_SP AT %MW62, 1 s
   "highoiltempsp" : Int = PLC oilhightemp_sp AT %MW60, 1 s
   "highoiltempdelay" : Int = PLC oilhighflowdelay_SP AT %MW58, 1 s
   "highoilflowdelay" : Int = PLC oilhighflowdelay_SP AT %MW58, 1 s
   "highoilflowsp" : Int = PLC oilhighflow_SP AT %MW70, 1 s
   "lowoilflowsp" : Int = PLC oillowflow_SP AT %MW44, 1 s
   "lowoilflowdelaysp" : Int = PLC oillowflowdelay_SP AT %MW46, 1 s
   "warmupoiltemp" : Int = PLC warmupoiltemp_SP AT %MW82, 1 s
   "warmupoildelay" : Int = PLC warmupoiltempdelay_sp AT %MW84, 1 s
   "currentsp" : Int = PLC stabilizekw_SPIN AT %MW92, 1 s
   "stabilizedelay" : Int = PLC stablizemode_delay AT %MW96, 1 s
   "cooldowntempsp" : Int = PLC cooldownoiltemp_sp AT %MW102, 1 s
   "cooldownoiltempdelay" : Int = PLC cooldowndelaysp AT %MW100, 1 s
   "vfdmaualSP" : Real = PLC vfdmanualsp AT %MD114, 1 s
   "bafflemanualSp" : Real = PLC bafflemanualsp AT %MD106, 1 s
   "generation_mode" : Bool = PLC generation_mode AT %M52.7, 1 s
   "warmupmode" : Bool = PLC warmup_mode AT %M52.3, 1 s
   "stabilizemode" : Bool = PLC stabilize_mode AT %M52.5, 1 s
   "idlemode" : Bool = PLC idlemode AT %M53.6, 1 s
   "cooldownmode" : Bool = PLC cooldown_mode AT %M53.1, 1 s
   "programlanguage" : Int = PLC PROGLANG AT %MW12, 1 s
   "LADPB" : Bool = PLC PB_LAD AT %M0.3, 1 s
   "FBDPB" : Bool = PLC PB_FBD AT %M1.0, 1 s
   "SCLPB" : Bool = PLC PB_SCL AT %M1.1, 1 s
   "STLPB" : Bool = PLC PB_STL AT %M1.2, 1 s
   "current" : Int = PLC curentout_SV AT %MW30, 1 s
   "oiltemp" : Int = PLC OiltempSV AT %MW24, 1 s
   "oilflow" : Int = PLC OilflowSV AT %MW26, 1 s
   "bafflepct" : Int = PLC baffle_pct AT %MW22, 1 s
   "vfdoilpumppct" : Int = PLC OilpumpVFD_pct AT %MW20, 1 s
   "rpm" : Int = PLC RPM_In AT %MW2, 1 s

screen "status" 640x480
   Circle "Circle_1" at 562,416 size 56x56
      Visibility <- "faultmode"
   TextField "Text field_1" at 564,431 size 54x22; Text 'Alarm!'
   Circle "Circle_2" at 561,416 size 56x56
      Visibility <- "faultmode"
   TextField "Text field_2" at 575,434 size 28x22; Text 'ok!'
   Button "Button_1" at 20,437 size 76x32; TextOff 'Main'
      on Click: ActivateScreen("status", 0)
   Button "Button_2" at 234,437 size 76x32; TextOff 'Alarms'
      on Click: ActivateScreen("Alarms", 0)
   Button "Button_3" at 354,438 size 76x32; TextOff 'config'
      on Click: ActivateScreen("Config", 0)
   Button "Button_4" at 127,438 size 76x32; TextOff 'Overview'
      on Click: ActivateScreen("Overview", 0)
   Group "Group_1" at 561,416 size 56x56
   Group "Group" at 562,416 size 56x56
   TextField "Text field_3" at 15,8 size 188x43; Text 'Mainscreen'
   TextField "Text field_4" at 392,39 size 224x38; Text 'Generation Mode'
      Visibility <- "generation_mode"
   TextField "Text field_5" at 424,39 size 192x38; Text 'Warmup Mode'
      Visibility <- "warmupmode"
   TextField "Text field_6" at 416,43 size 190x38; Text 'stabilize Mode'
      Visibility <- "stabilizemode"
   TextField "Text field_7" at 408,39 size 137x38; Text 'Idle mode'
      Visibility <- "idlemode"
   TextField "Text field_8" at 410,39 size 208x38; Text 'Cooldown Mode'
      Visibility <- "cooldownmode"
   Button "Button_5" at 40,241 size 57x32; TextOff 'LAD'
      on Press: SetBit("LADPB")
      on Release: ResetBit("LADPB")
   Button "Button_6" at 145,238 size 57x32; TextOff 'FBD'
      on Release: ResetBit("FBDPB")
      on Press: SetBit("FBDPB")
   Button "Button_7" at 37,293 size 57x32; TextOff 'SCL'
      on Release: ResetBit("SCLPB")
      on Press: SetBit("SCLPB")
   Button "Button_8" at 142,296 size 57x32; TextOff 'STL'
      on Release: ResetBit("STLPB")
      on Press: SetBit("STLPB")
   Button "Button_9" at 425,90 size 165x32; TextOff 'LADDER LOGIC'
      Visibility <- "programlanguage"
   Button "Button_10" at 430,90 size 165x32; TextOff 'FUNCTION BLOCK'
      Visibility <- "programlanguage"
   Button "Button_11" at 410,92 size 196x32; TextOff 'STRUCTURED CONTROL'
      Visibility <- "programlanguage"
   Button "Button_12" at 428,92 size 165x32; TextOff 'STATEMENT LIST'
      Visibility <- "programlanguage"
   Button "Button_13" at 26,372 size 134x32; TextOff 'START'
      on Click: ActivateScreen("status", 0)
      on Press: SetBit("systemstart_pb")
      on Release: ResetBit("systemstart_pb")
   Button "Button_14" at 178,372 size 132x32; TextOff 'STOP'
      on Click: ActivateScreen("status", 0)
      on Press: SetBit("systemstop_pb")
      on Release: ResetBit("systemstop_pb")
      Visibility <- "generation_mode"
   IOField "I/O field_1" at 165,79 size 102x38; FormatPattern s99999
      ProcessValue <- "current"
   TextField "Text field_9" at 16,75 size 128x39; Text 'Current:'
   TextField "Text field_10" at 281,81 size 45x37; Text 'kw'
   TextField "Text field_11" at 3,121 size 150x39; Text 'Interlock:'
   Button "Button_15" at 165,122 size 119x42; TextOff 'Engaged'
      Visibility <- "stationinterlockEn"
   Button "Button_16" at 165,124 size 119x42; TextOff 'Offline'
   IOField "I/O field_2" at 488,182 size 81x38; FormatPattern s99999
      ProcessValue <- "HM_minutes"
   IOField "I/O field_3" at 488,234 size 79x38; FormatPattern s99999
      ProcessValue <- "HM_hours"
   IOField "I/O field_4" at 488,286 size 83x38; FormatPattern s99999
      ProcessValue <- "HM_days"
   TextField "Text field_12" at 350,180 size 122x39; Text 'Minutes'
   TextField "Text field_13" at 375,234 size 92x39; Text 'Hours'
   TextField "Text field_14" at 387,282 size 76x39; Text 'Days'
   Button "Button_17" at 409,337 size 132x32; TextOff 'Hourmeter Reset'
      on Click: ActivateScreen("status", 0)
      on Release: ResetBit("hourmetereset_pb")
      on Press: SetBit("hourmetereset_pb")
      Visibility <- "generation_mode"
   TextField "Text field_15" at 394,134 size 164x39; Text 'Hourmeter'
   TextField "Text field_16" at 9,175 size 258x39; Text 'Select Paradaigm'
   Button "Button_18" at 458,435 size 76x32; TextOff 'Exit'
      on Click: StopRuntime(0)

screen "Overview" 640x480
   Button "Button_1" at 20,437 size 76x32; TextOff 'Main'
      on Click: ActivateScreen("status", 0)
   Button "Button_2" at 262,437 size 76x32; TextOff 'Alarms'
      on Click: ActivateScreen("Alarms", 0)
   Button "Button_3" at 380,437 size 76x32; TextOff 'config'
      on Click: ActivateScreen("Config", 0)
   Button "Button_4" at 140,437 size 76x32; TextOff 'Overview'
      on Click: ActivateScreen("Overview", 0)
   TextField "Text field_3" at 15,8 size 158x43; Text 'Overview'
   GraphicView "Graphic view_1" at -32,89 size 696x264; Picture "Capture"
      Visibility <- "brakeEn"
   TextField "Text field_4" at 15,3 size 158x43; Text 'Overview'
   TextField "Text field_5" at 12,181 size 50x22; Text 'Baffle'
   TextField "Text field_6" at 109,191 size 87x22; Text 'Alarm horn'
   TextField "Text field_7" at 256,181 size 81x22; Text 'Generator'
   TextField "Text field_8" at 375,136 size 68x22; Text 'oil pump'
   TextField "Text field_9" at 514,88 size 111x22; Text 'Power Station'
   IOField "I/O field_1" at 12,311 size 55x32; FormatPattern 9999999
      ProcessValue <- "bafflepct"
   TextField "Text field_10" at 12,353 size 81x25; Text 'Baffle %'
   IOField "I/O field_2" at 334,311 size 55x32; FormatPattern 9999999
      ProcessValue <- "rpm"
   TextField "Text field_11" at 334,354 size 43x25; Text 'RPM'
   IOField "I/O field_3" at 262,94 size 55x32; FormatPattern 9999999
      ProcessValue <- "vfdoilpumppct"
   TextField "Text field_12" at 245,131 size 102x25; Text 'Oilpump %'
   Group "Group_2" at 413,311 size 145x37
   Group "Group_3" at 411,311 size 147x37
   Group "Group_4" at 33,57 size 147x37
   Group "Group_5" at 34,57 size 147x37
   TextField "Text field_21" at 2,52 size 224x38; Text 'Generation Mode'
      Visibility <- "generation_mode"
   TextField "Text field_22" at 34,52 size 192x38; Text 'Warmup Mode'
      Visibility <- "warmupmode"
   TextField "Text field_23" at 26,56 size 190x38; Text 'stabilize Mode'
      Visibility <- "stabilizemode"
   TextField "Text field_24" at 18,52 size 137x38; Text 'Idle mode'
      Visibility <- "idlemode"
   TextField "Text field_25" at 2,57 size 208x38; Text 'Cooldown Mode'
      Visibility <- "cooldownmode"
   Group "Group_1" at 561,416 size 56x56
   Group "Group" at 562,416 size 56x56
   Rectangle "Rectangle_1" at 413,311 size 145x37
      Visibility <- "brakeEn"
   TextField "Text field_14" at 417,318 size 132x22; Text 'BRAKE ENGAGED'
      Visibility <- "brakeEn"
   Rectangle "Rectangle_2" at 411,311 size 147x37
      Visibility <- "brakeEn"
   TextField "Text field_15" at 415,318 size 137x22; Text 'BRAKE RELEASED'
      Visibility <- "brakeEn"
   Rectangle "Rectangle_3" at 33,57 size 147x37
      Visibility <- "stationinterlockEn"
   TextField "Text field_16" at 37,64 size 141x22; Text 'Interlock Engaged'
      Visibility <- "stationinterlockEn"
   Rectangle "Rectangle_4" at 34,57 size 147x37
      Visibility <- "stationinterlockEn"
   TextField "Text field_17" at 58,64 size 99x22; Text 'No Interlock'
      Visibility <- "stationinterlockEn"
   Circle "Circle_2" at 561,416 size 56x56
      Visibility <- "faultmode"
   TextField "Text field_2" at 575,434 size 28x22; Text 'ok!'
   Circle "Circle_1" at 562,416 size 56x56
      Visibility <- "faultmode"
   TextField "Text field_1" at 564,431 size 54x22; Text 'Alarm!'

screen "Alarms" 640x480
   Button "Button_1" at 20,437 size 76x32; TextOff 'Main'
      on Click: ActivateScreen("status", 0)
   Button "Button_2" at 262,437 size 76x32; TextOff 'Alarms'
      on Click: ActivateScreen("Alarms", 0)
   Button "Button_3" at 380,437 size 76x32; TextOff 'config'
      on Click: ActivateScreen("Config", 0)
   Button "Button_4" at 140,437 size 76x32; TextOff 'Overview'
      on Click: ActivateScreen("Overview", 0)
   TextField "Text field_3" at 18,7 size 117x43; Text 'Alarms'
   Button "Button_5" at 20,294 size 135x32; TextOff 'ALARM RESET'
      on Press: SetBit("alarmreset")
      on Release: ResetBit("alarmreset")
   Button "Button_6" at 447,294 size 151x32; TextOff 'ALARM SIELNCE'
      on Press: SetBit("alarmsilence")
      on Release: ResetBit("alarmsilence")
   Group "Group_2" at 20,340 size 58x58
   Group "Group_3" at 94,339 size 59x59
   Group "Group_4" at 168,338 size 60x60
   Group "Group_5" at 240,336 size 66x62
   Group "Group_6" at 315,335 size 64x63
   Group "Group_7" at 391,340 size 62x57
   Group "Group_8" at 464,337 size 64x61
   Group "Group_9" at 14,333 size 546x80
   Group "Group_1" at 561,416 size 56x56
   Group "Group" at 562,416 size 56x56
   AlarmView "Alarm view_1" at 29,54 size 556x234
   Circle "Circle_3" at 20,340 size 58x58
      Visibility <- "E-stop_alarm"
   TextField "Text field_4" at 22,357 size 55x22; Text 'ESTOP'
   Circle "Circle_4" at 94,339 size 59x59
      Visibility <- "brakefailurealarm"
   TextField "Text field_5" at 94,358 size 55x22; Text 'BRAKE'
   Circle "Circle_5" at 168,338 size 60x60
      Visibility <- "overspeedalarm"
   TextField "Text field_6" at 171,358 size 54x22; Text 'SPEED'
   Circle "Circle_6" at 240,336 size 62x62
      Visibility <- "highoilflow_alarm"
   TextField "Text field_7" at 240,358 size 66x22; Text 'H.FLOW'
   Circle "Circle_7" at 316,335 size 63x63
      Visibility <- "lowoilflow_alarm"
   TextField "Text field_8" at 315,358 size 64x22; Text 'L.FLOW'
   Circle "Circle_8" at 394,340 size 57x57
      Visibility <- "highoiltemp_alarm"
   TextField "Text field_9" at 391,359 size 62x22; Text 'H.TEMP'
   Circle "Circle_9" at 464,337 size 61x61
      Visibility <- "overcurrentalarm"
   TextField "Text field_10" at 464,360 size 64x22; Text 'O.CRNT'
   Rectangle "Rectangle_1" at 14,333 size 546x80
      Visibility <- "faultmode"
   TextField "Text field_11" at 227,360 size 130x29; Text 'NO ALARMS'
   Circle "Circle_2" at 561,416 size 56x56
      Visibility <- "faultmode"
   TextField "Text field_2" at 575,434 size 28x22; Text 'ok!'
   Circle "Circle_1" at 562,416 size 56x56
      Visibility <- "faultmode"
   TextField "Text field_1" at 564,431 size 54x22; Text 'Alarm!'

screen "Config" 640x480
   Button "Button_1" at 20,437 size 76x32; TextOff 'Main'
      on Click: ActivateScreen("status", 0)
   Button "Button_2" at 262,437 size 76x32; TextOff 'Alarms'
      on Click: ActivateScreen("Alarms", 0)
   Button "Button_3" at 380,437 size 76x32; TextOff 'config'
      on Click: ActivateScreen("Config", 0)
   Button "Button_4" at 140,437 size 76x32; TextOff 'Overview'
      on Click: ActivateScreen("Overview", 0)
   TextField "Text field_3" at 15,8 size 224x43; Text 'Configuration'
   IOField "I/O field_1" at 160,107 size 57x24; FormatPattern s99999
      ProcessValue <- "warmupoiltemp"
   TextField "Text field_4" at 23,50 size 176x34; Text 'Process value'
   TextField "Text field_5" at 16,111 size 129x25; Text 'Warmup Temp'
   TextField "Text field_6" at 21,149 size 128x25; Text 'Warmup delay'
   TextField "Text field_7" at 20,184 size 127x25; Text 'stabilize delay'
   TextField "Text field_8" at 22,216 size 120x25; Text 'Current (kw)'
   TextField "Text field_9" at 6,250 size 141x25; Text 'cooldown Temp'
   TextField "Text field_10" at 9,281 size 140x25; Text 'cooldown delay'
   IOField "I/O field_2" at 159,147 size 57x26; FormatPattern s99999
      ProcessValue <- "warmupoildelay"
   IOField "I/O field_3" at 158,183 size 57x24; FormatPattern s99999
      ProcessValue <- "stabilizedelay"
   IOField "I/O field_4" at 158,216 size 57x24; FormatPattern s99999
      ProcessValue <- "current"
   IOField "I/O field_5" at 160,245 size 57x27; FormatPattern 9999999
      ProcessValue <- "cooldowntempsp"
   IOField "I/O field_6" at 159,281 size 57x25; FormatPattern s99999
      ProcessValue <- "cooldownoiltempdelay"
   IOField "I/O field_7" at 588,67 size 52x24; FormatPattern s99999
      ProcessValue <- "lowoilflowsp"
   TextField "Text field_11" at 344,17 size 155x34; Text 'Alarm value'
   TextField "Text field_12" at 456,159 size 130x25; Text 'low flow delay'
   TextField "Text field_13" at 457,71 size 123x25; Text 'low flow GPM'
   TextField "Text field_14" at 235,96 size 158x25; Text 'Overcurrent delay'
   TextField "Text field_18" at 257,65 size 132x25; Text 'Overcurrent sp'
   TextField "Text field_15" at 451,188 size 139x25; Text 'High flow delay'
   TextField "Text field_16" at 456,98 size 132x25; Text 'High flow GPM'
   TextField "Text field_17" at 239,124 size 152x25; Text 'Over speed delay'
   TextField "Text field_19" at 451,130 size 137x25; Text 'overspeed RPM'
   TextField "Text field_20" at 229,189 size 164x25; Text 'oilhigh temp delay'
   TextField "Text field_21" at 246,217 size 143x25; Text 'oil high temp sp'
   TextField "Text field_22" at 232,154 size 164x25; Text 'brake failure delay'
   IOField "I/O field_8" at 587,130 size 52x24; FormatPattern s99999
      ProcessValue <- "overcurrrentsp"
   IOField "I/O field_9" at 398,67 size 52x24; FormatPattern s99999
      ProcessValue <- "overcurrrentsp"
   IOField "I/O field_10" at 398,96 size 52x24; FormatPattern s99999
      ProcessValue <- "overcurrentdelay"
   IOField "I/O field_11" at 587,98 size 52x24; FormatPattern s99999
      ProcessValue <- "highoilflowsp"
   IOField "I/O field_12" at 586,189 size 52x24; FormatPattern s99999
      ProcessValue <- "highoilflowdelay"
   IOField "I/O field_13" at 399,126 size 52x24; FormatPattern s99999
      ProcessValue <- "overspeeddelay"
   IOField "I/O field_14" at 398,157 size 52x24; FormatPattern s99999
      ProcessValue <- "brakefailuredelay"
   IOField "I/O field_15" at 398,188 size 52x24; FormatPattern s99999
      ProcessValue <- "highoiltempdelay"
   IOField "I/O field_16" at 398,217 size 52x24; FormatPattern s99999
      ProcessValue <- "highoiltempsp"
   IOField "I/O field_18" at 587,162 size 52x24; FormatPattern s99999
      ProcessValue <- "lowoilflowdelaysp"
   TextField "Text field_23" at 533,317 size 102x25; Text 'Alarm Horn'
   TextField "Text field_24" at 443,319 size 54x25; Text 'Brake'
   TextField "Text field_25" at 266,318 size 152x25; Text 'Station InterlocK'
   TextField "Text field_26" at 158,319 size 56x25; Text 'Baffle'
   TextField "Text field_27" at 3,318 size 114x25; Text 'oilpump VFD'
   TextField "Text field_28" at 309,280 size 172x29; Text 'HOA CONTROLS'
   Button "Button_5" at 533,345 size 26x25; TextOff 'H'
      on Press: SetBit("alarmhornhandpb")
      on Release: ResetBit("alarmhornhandpb")
   Button "Button_6" at 567,345 size 26x25; TextOff 'O'
      on Press: SetBit("alarmhornoffpb")
      on Release: ResetBit("alarmhornoffpb")
   Button "Button_7" at 598,345 size 26x25; TextOff 'A'
      on Release: ResetBit("alarmhornautopb")
      on Press: SetBit("alarmhornautopb")
   Rectangle "Rectangle_4" at 566,380 size 28x24
      Visibility <- "alarmhornhoa"
   Rectangle "Rectangle_5" at 566,379 size 28x24
      Visibility <- "alarmhornhoa"
   Rectangle "Rectangle_6" at 566,379 size 28x24
      Visibility <- "alarmhornhoa"
   Rectangle "Rectangle_7" at 9,379 size 28x24
      Visibility <- "vfdhoa"
   Rectangle "Rectangle_8" at 8,379 size 28x24
      Visibility <- "vfdhoa"
   Rectangle "Rectangle_9" at 8,379 size 28x24
      Visibility <- "vfdhoa"
   Rectangle "Rectangle_10" at 144,379 size 28x24
      Visibility <- "bafflehoa"
   Rectangle "Rectangle_11" at 144,380 size 28x24
      Visibility <- "bafflehoa"
   Rectangle "Rectangle_12" at 144,380 size 28x24
      Visibility <- "bafflehoa"
   Rectangle "Rectangle_13" at 324,383 size 28x24
      Visibility <- "stationinterlockhoa"
   Rectangle "Rectangle_14" at 323,383 size 28x24
      Visibility <- "stationinterlockhoa"
   Rectangle "Rectangle_15" at 324,382 size 28x24
      Visibility <- "stationinterlockhoa"
   Rectangle "Rectangle_16" at 461,383 size 28x24
      Visibility <- "brakehoa"
   Rectangle "Rectangle_17" at 461,383 size 28x24
      Visibility <- "brakehoa"
   Rectangle "Rectangle_18" at 462,383 size 28x24
      Visibility <- "brakehoa"
   Button "Button_8" at 424,349 size 26x25; TextOff 'H'
      on Release: ResetBit("brakehandpb")
      on Press: SetBit("brakehandpb")
   Button "Button_9" at 458,349 size 26x25; TextOff 'O'
      on Release: ResetBit("brakeoffpb")
      on Press: SetBit("brakeoffpb")
   Button "Button_10" at 489,349 size 26x25; TextOff 'A'
      on Release: ResetBit("brakeautopb")
      on Press: SetBit("brakeautopb")
   Button "Button_11" at 284,349 size 26x25; TextOff 'H'
      on Release: ResetBit("stationinterlockhandpb")
      on Press: SetBit("stationinterlockhandpb")
   Button "Button_12" at 322,348 size 26x25; TextOff 'O'
      on Release: ResetBit("stationinterlockoffpb")
      on Press: SetBit("stationinterlockoffpb")
   Button "Button_13" at 361,348 size 26x25; TextOff 'A'
      on Release: ResetBit("stationinterlockautopb")
      on Press: SetBit("stationinterlockautopb")
   Button "Button_14" at 140,349 size 26x25; TextOff 'H'
      on Release: ResetBit("bafflehandpb")
      on Press: SetBit("bafflehandpb")
   Button "Button_15" at 172,350 size 26x25; TextOff 'O'
      on Release: ResetBit("baffleoffpb")
      on Press: SetBit("baffleoffpb")
   Button "Button_16" at 204,349 size 26x25; TextOff 'A'
      on Release: ResetBit("baffleautopb")
      on Press: SetBit("baffleautopb")
   Button "Button_17" at 9,347 size 26x25; TextOff 'H'
      on Release: ResetBit("vfdhandpb")
      on Press: SetBit("vfdhandpb")
   Button "Button_18" at 39,347 size 26x25; TextOff 'O'
      on Release: ResetBit("vfdoffpb")
      on Press: SetBit("vfdoffpb")
   Button "Button_19" at 70,347 size 26x25; TextOff 'A'
      on Release: ResetBit("vfdautopb")
      on Press: SetBit("vfdautopb")
   IOField "I/O field_17" at 74,381 size 51x25; FormatPattern s999999999.999
      ProcessValue <- "vfdmaualSP"
   TextField "Text field_29" at 43,382 size 27x25; Text 'SP'
   IOField "I/O field_19" at 205,379 size 51x25; FormatPattern s999999999.999
      ProcessValue <- "bafflemanualSp"
   TextField "Text field_30" at 177,380 size 27x25; Text 'SP'
   Group "Group_1" at 561,416 size 56x56
   Group "Group" at 562,416 size 56x56
   Circle "Circle_2" at 561,416 size 56x56
      Visibility <- "faultmode"
   TextField "Text field_2" at 575,434 size 28x22; Text 'ok!'
   Circle "Circle_1" at 562,416 size 56x56
      Visibility <- "faultmode"
   TextField "Text field_1" at 564,431 size 54x22; Text 'Alarm!'
*)